KUKA KRL data list: kuka_eki_ros_sub.dat

&ACCESS RVO
defdat kuka_eki_ros_sub
   ext bas(bas_command  :in,real  :in )
enddat
